// A helper class providing various helpful methods when working with ams data
PROGRAM AmsHelper
VAR
END_VAR

// Converts netId of type <Tc2_System.T_AmsNetIdArr> to <T_AmsNetID>, which equates to <STRING(23)>.
METHOD PUBLIC NetIdToString : T_AmsNetID
VAR_INPUT
	netId	: Tc2_System.T_AmsNetIdArr;	// NetId to be converted
END_VAR

VAR
	arrayMaxIndex	: DINT;
	i				: DINT;
END_VAR
arrayMaxIndex := ArrayHelper.GetMaxIndex(arr := netId, dataType := netId[0], startIndex := 0);

FOR i := 0 TO arrayMaxIndex BY 1 DO
	IF netId[i] <> 0 THEN
		EXIT;
	END_IF
	IF i = ArrayHelper.GetMaxIndex(arr := netId, dataType := netId[0], startIndex := 0) THEN
		NetIdToString := '';
		RETURN;
	END_IF
END_FOR

NetIdToString := Tc2_System.F_CreateAmsNetId(nIds := netId);
END_METHOD

END_PROGRAM

(* stored: Version 1.1.0.1, ProductVersion 3.1.4024.13
   POU AmsHelper: Id {6d6b745e-a376-00e4-05e8-9f698802219e}, SpecialFunc None
   Method NetIdToString: Id {6a8678c3-457e-04b0-30f5-773ba24b8108} *)
